# EPICS substitutions: dg645App/Db/regens.substitutions
file regens.template {
pattern
{REG, CHAN1, CHAN2}
{  1,     4,     5}
{  2,     6,     7}
{  3,     8,     9}
}
